% RSLogix 500 project T4150574.RSS, saved by version 8.10.00.18 %
PROJECT "T4150574"    % processor: SLC 500, 1747-L542 %

PROGRAM FILES
  LAD 2   89 rungs
  LAD 3   93 rungs
  LAD 4   69 rungs
  LAD 5   3 rungs
  LAD 6   136 rungs
  LAD 9   34 rungs
  LAD 10   90 rungs
  LAD 11   20 rungs
  LAD 12   13 rungs
  LAD 15   61 rungs
  LAD 16   27 rungs
  LAD 17   7 rungs
  LAD 18   55 rungs
  LAD 21   5 rungs
  LAD 22   82 rungs
  LAD 23   74 rungs
  LAD 24   136 rungs
  LAD 26   178 rungs
  LAD 27   27 rungs
  LAD 28   29 rungs
  LAD 31   238 rungs
  LAD 36   69 rungs
  LAD 41   9 rungs
  LAD 50   338 rungs
  LAD 51   183 rungs
  LAD 52   5 rungs
  LAD 53   6 rungs
  LAD 60   11 rungs
  LAD 71   9 rungs
  LAD 75   5 rungs
  LAD 76   5 rungs
  LAD 77   5 rungs
  LAD 78   6 rungs
  LAD 80   7 rungs
  LAD 120   43 rungs
  LAD 126   33 rungs
  LAD 127   30 rungs
  LAD 129   29 rungs
  LAD 131   44 rungs
  LAD 132   40 rungs
  LAD 133   25 rungs
  LAD 134   25 rungs

DATA FILES
  O0 OUTPUT  58 elements
  I1 INPUT  52 elements
  S2 STATUS  164 elements
  B3 BINARY  150 elements
  T4 TIMER  122 elements
  C5 COUNTER  6 elements
  R6 CONTROL  20 elements
  N7 INTEGER  53 elements
  F8 FLOAT  50 elements
  N9   14 elements
  B10   12 elements
  B11   33 elements
  B12   14 elements
  B15   1 elements
  B16   5 elements
  B17   5 elements
  B18   4 elements
  T21   85 elements
  B22   12 elements
  B23   8 elements
  B24   8 elements
  N25   195 elements
  B28   10 elements
  B29   15 elements
  B30   1 elements
  T31   50 elements
  N32   137 elements
  B35   9 elements
  B36   2 elements
  N40   240 elements
  N41   240 elements
  N42   240 elements
  N43   240 elements
  N44   240 elements
  N45   240 elements
  N46   240 elements
  N47   240 elements
  N48   120 elements
  B49   50 elements
  N50   60 elements
  N51   256 elements
  N52   100 elements
  B53   100 elements
  N54   100 elements
  N60   214 elements
  N61   250 elements
  N62   250 elements
  N63   250 elements
  N75   200 elements
  N76   50 elements
  N77   100 elements
  N78   50 elements
  N79   50 elements
  B84   4 elements
  N89   200 elements
  N90   20 elements
  N91   250 elements
  N92   250 elements
  N93   250 elements
  N94   250 elements
  N95   250 elements
  N100   50 elements
  N105   20 elements
  N110   80 elements

LADDER 2
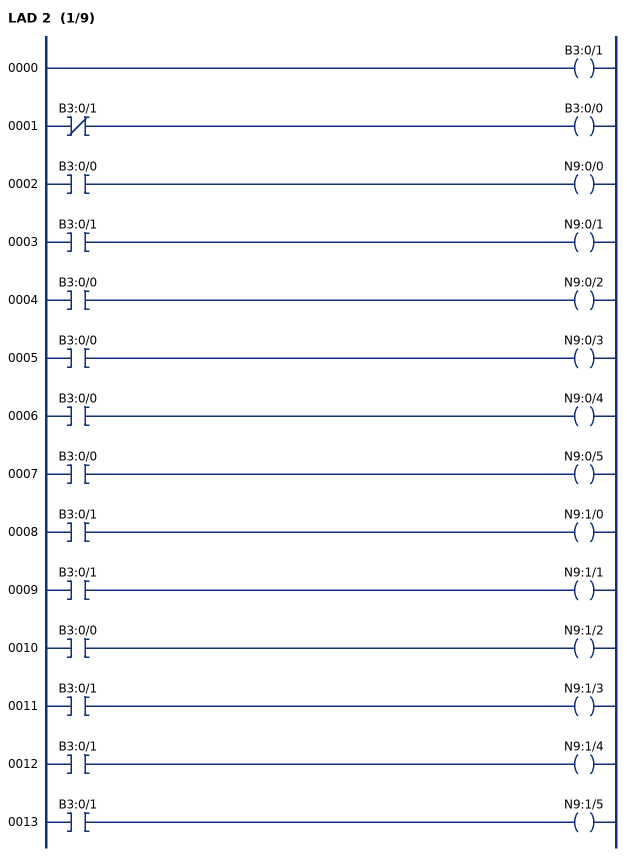
% Rung: 0 %
SOR OTE B3:0/1 EOR
% Rung: 1 %
SOR XIO B3:0/1 OTE B3:0/0 EOR
% Rung: 2 %
SOR XIC B3:0/0 OTE N9:0/0 EOR
% Rung: 3 %
SOR XIC B3:0/1 OTE N9:0/1 EOR
% Rung: 4 %
SOR XIC B3:0/0 OTE N9:0/2 EOR
% Rung: 5 %
SOR XIC B3:0/0 OTE N9:0/3 EOR
% Rung: 6 %
SOR XIC B3:0/0 OTE N9:0/4 EOR
% Rung: 7 %
SOR XIC B3:0/0 OTE N9:0/5 EOR
% Rung: 8 %
SOR XIC B3:0/1 OTE N9:1/0 EOR
% Rung: 9 %
SOR XIC B3:0/1 OTE N9:1/1 EOR
% Rung: 10 %
SOR XIC B3:0/0 OTE N9:1/2 EOR
% Rung: 11 %
SOR XIC B3:0/1 OTE N9:1/3 EOR
% Rung: 12 %
SOR XIC B3:0/1 OTE N9:1/4 EOR
% Rung: 13 %
SOR XIC B3:0/1 OTE N9:1/5 EOR

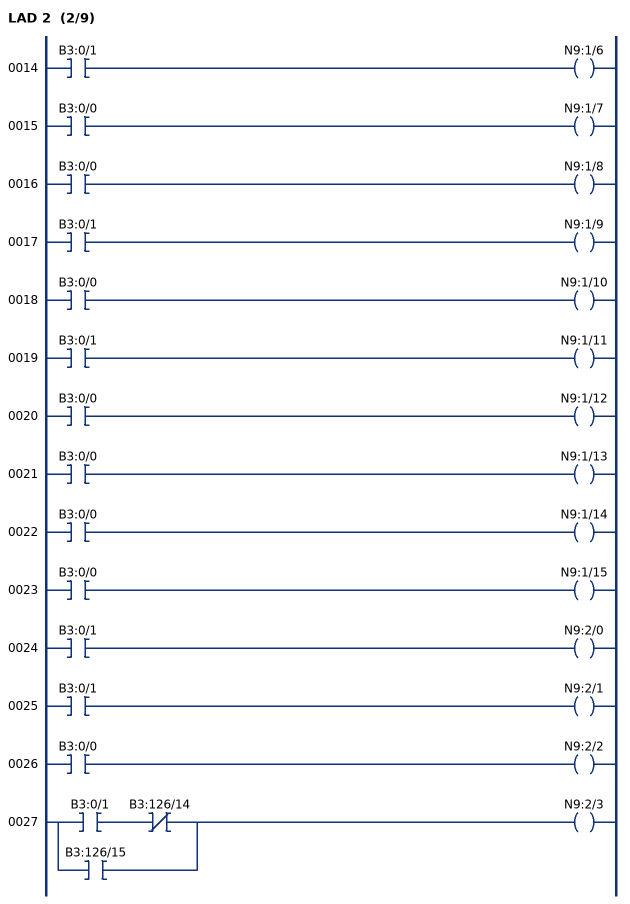
% Rung: 14 %
SOR XIC B3:0/1 OTE N9:1/6 EOR
% Rung: 15 %
SOR XIC B3:0/0 OTE N9:1/7 EOR
% Rung: 16 %
SOR XIC B3:0/0 OTE N9:1/8 EOR
% Rung: 17 %
SOR XIC B3:0/1 OTE N9:1/9 EOR
% Rung: 18 %
SOR XIC B3:0/0 OTE N9:1/10 EOR
% Rung: 19 %
SOR XIC B3:0/1 OTE N9:1/11 EOR
% Rung: 20 %
SOR XIC B3:0/0 OTE N9:1/12 EOR
% Rung: 21 %
SOR XIC B3:0/0 OTE N9:1/13 EOR
% Rung: 22 %
SOR XIC B3:0/0 OTE N9:1/14 EOR
% Rung: 23 %
SOR XIC B3:0/0 OTE N9:1/15 EOR
% Rung: 24 %
SOR XIC B3:0/1 OTE N9:2/0 EOR
% Rung: 25 %
SOR XIC B3:0/1 OTE N9:2/1 EOR
% Rung: 26 %
SOR XIC B3:0/0 OTE N9:2/2 EOR
% Rung: 27 %
SOR BST XIC B3:0/1 XIO B3:126/14 NXB XIC B3:126/15 BND OTE N9:2/3 EOR

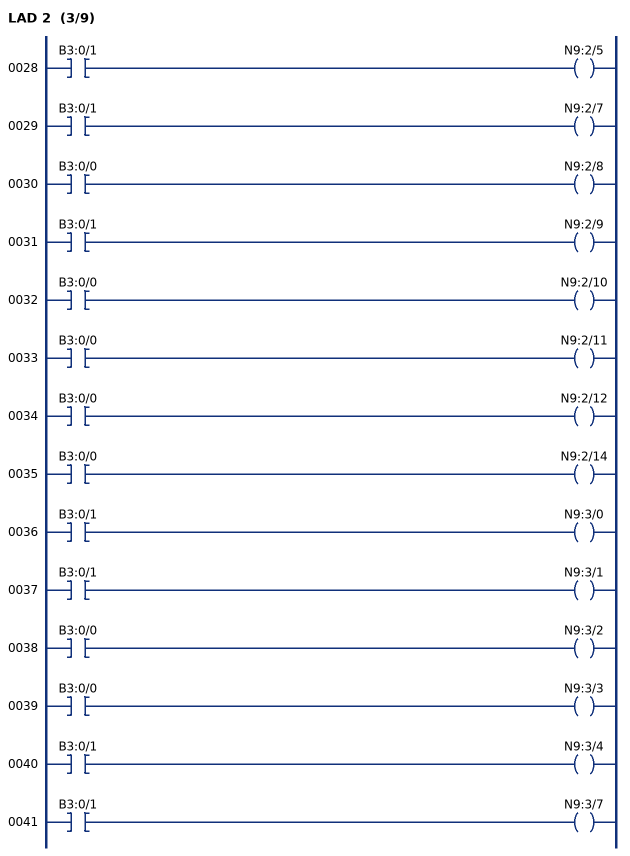
% Rung: 28 %
SOR XIC B3:0/1 OTE N9:2/5 EOR
% Rung: 29 %
SOR XIC B3:0/1 OTE N9:2/7 EOR
% Rung: 30 %
SOR XIC B3:0/0 OTE N9:2/8 EOR
% Rung: 31 %
SOR XIC B3:0/1 OTE N9:2/9 EOR
% Rung: 32 %
SOR XIC B3:0/0 OTE N9:2/10 EOR
% Rung: 33 %
SOR XIC B3:0/0 OTE N9:2/11 EOR
% Rung: 34 %
SOR XIC B3:0/0 OTE N9:2/12 EOR
% Rung: 35 %
SOR XIC B3:0/0 OTE N9:2/14 EOR
% Rung: 36 %
SOR XIC B3:0/1 OTE N9:3/0 EOR
% Rung: 37 %
SOR XIC B3:0/1 OTE N9:3/1 EOR
% Rung: 38 %
SOR XIC B3:0/0 OTE N9:3/2 EOR
% Rung: 39 %
SOR XIC B3:0/0 OTE N9:3/3 EOR
% Rung: 40 %
SOR XIC B3:0/1 OTE N9:3/4 EOR
% Rung: 41 %
SOR XIC B3:0/1 OTE N9:3/7 EOR

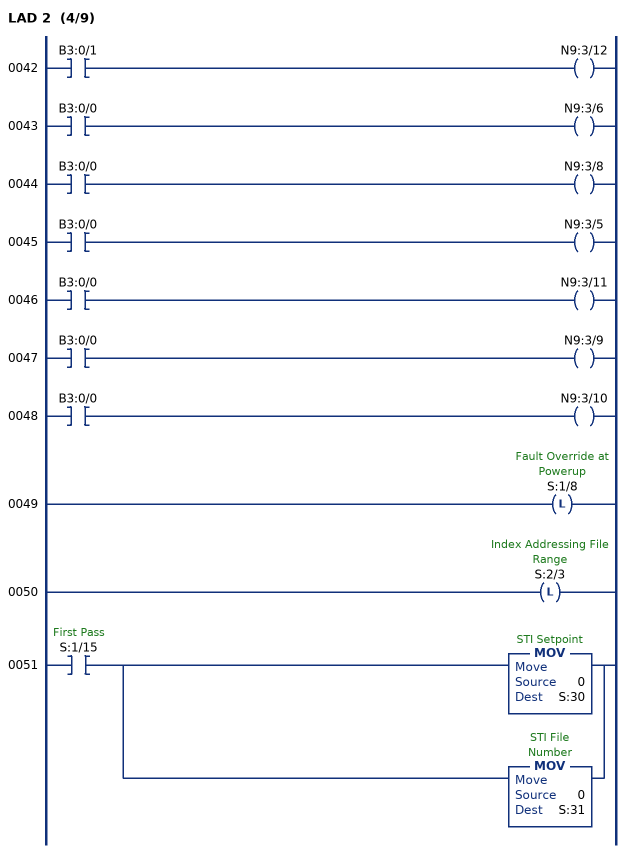
% Rung: 42 %
SOR XIC B3:0/1 OTE N9:3/12 EOR
% Rung: 43 %
SOR XIC B3:0/0 OTE N9:3/6 EOR
% Rung: 44 %
SOR XIC B3:0/0 OTE N9:3/8 EOR
% Rung: 45 %
SOR XIC B3:0/0 OTE N9:3/5 EOR
% Rung: 46 %
SOR XIC B3:0/0 OTE N9:3/11 EOR
% Rung: 47 %
SOR XIC B3:0/0 OTE N9:3/9 EOR
% Rung: 48 %
SOR XIC B3:0/0 OTE N9:3/10 EOR
% Rung: 49 %
SOR OTL S:1/8 EOR
%   S:1/8  "Fault Override at Powerup" %
% Rung: 50 %
SOR OTL S:2/3 EOR
%   S:2/3  "Index Addressing File Range" %
% Rung: 51 %
SOR XIC S:1/15 BST MOV 0 S:30 NXB MOV 0 S:31 BND EOR
%   S:1/15  "First Pass" %
%   S:30  "STI Setpoint" %
%   S:31  "STI File Number" %

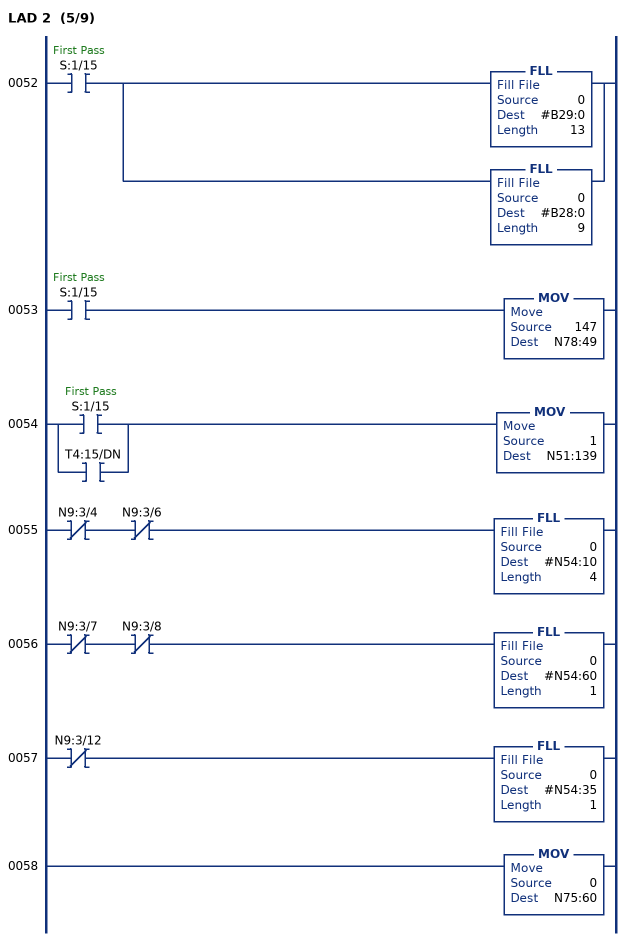
% Rung: 52 %
SOR XIC S:1/15 BST FLL 0 #B29:0 13 NXB FLL 0 #B28:0 9 BND EOR
%   S:1/15  "First Pass" %
% Rung: 53 %
SOR XIC S:1/15 MOV 147 N78:49 EOR
%   S:1/15  "First Pass" %
% Rung: 54 %
SOR BST XIC S:1/15 NXB XIC T4:15/DN BND MOV 1 N51:139 EOR
%   S:1/15  "First Pass" %
% Rung: 55 %
SOR XIO N9:3/4 XIO N9:3/6 FLL 0 #N54:10 4 EOR
% Rung: 56 %
SOR XIO N9:3/7 XIO N9:3/8 FLL 0 #N54:60 1 EOR
% Rung: 57 %
SOR XIO N9:3/12 FLL 0 #N54:35 1 EOR
% Rung: 58 %
SOR MOV 0 N75:60 EOR

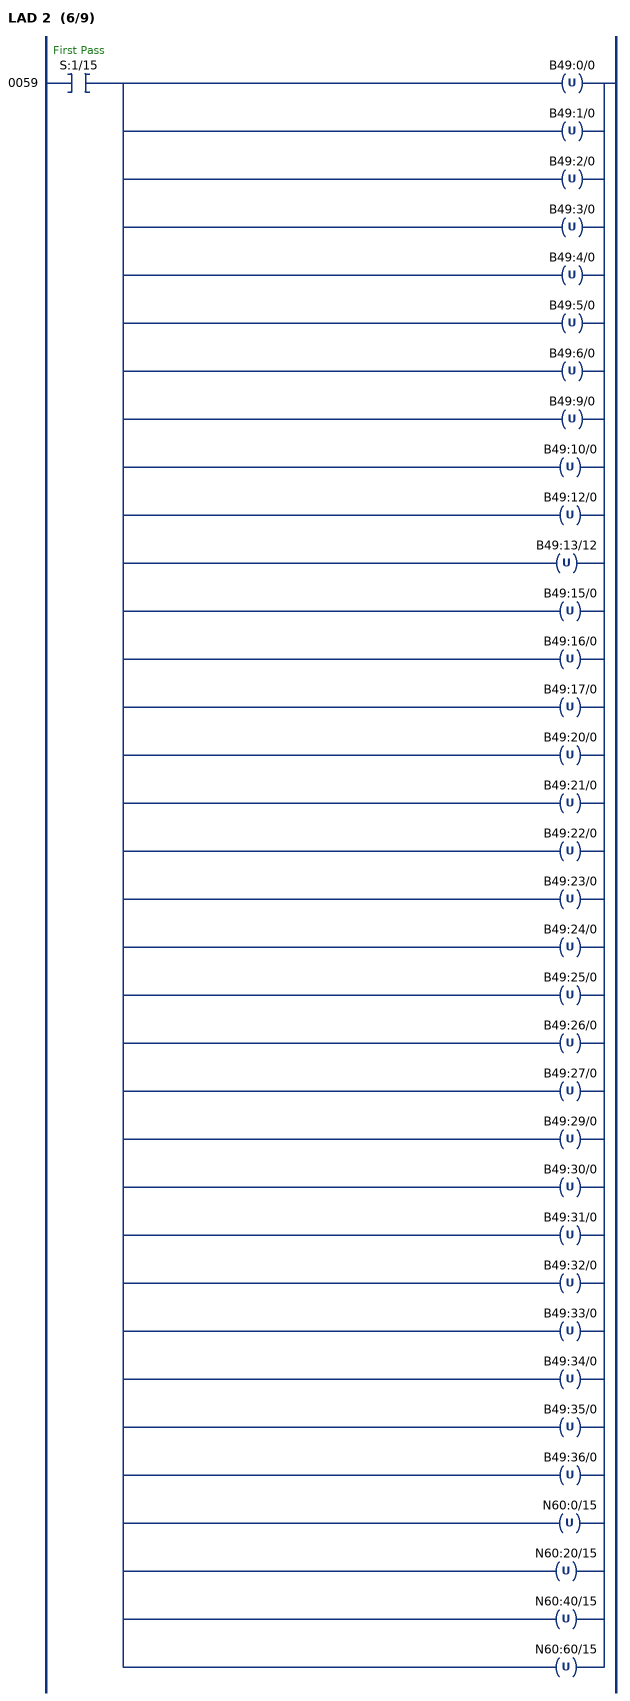
% Rung: 59 %
SOR XIC S:1/15 BST OTU B49:0/0 NXB OTU B49:1/0 NXB OTU B49:2/0 NXB OTU B49:3/0 NXB OTU B49:4/0 NXB OTU B49:5/0 NXB OTU B49:6/0 NXB OTU B49:9/0 NXB OTU B49:10/0 NXB OTU B49:12/0 NXB OTU B49:13/12 NXB OTU B49:15/0 NXB OTU B49:16/0 NXB OTU B49:17/0 NXB OTU B49:20/0 NXB OTU B49:21/0 NXB OTU B49:22/0 NXB OTU B49:23/0 NXB OTU B49:24/0 NXB OTU B49:25/0 NXB OTU B49:26/0 NXB OTU B49:27/0 NXB OTU B49:29/0 NXB OTU B49:30/0 NXB OTU B49:31/0 NXB OTU B49:32/0 NXB OTU B49:33/0 NXB OTU B49:34/0 NXB OTU B49:35/0 NXB OTU B49:36/0 NXB OTU N60:0/15 NXB OTU N60:20/15 NXB OTU N60:40/15 NXB OTU N60:60/15 BND EOR
%   S:1/15  "First Pass" %

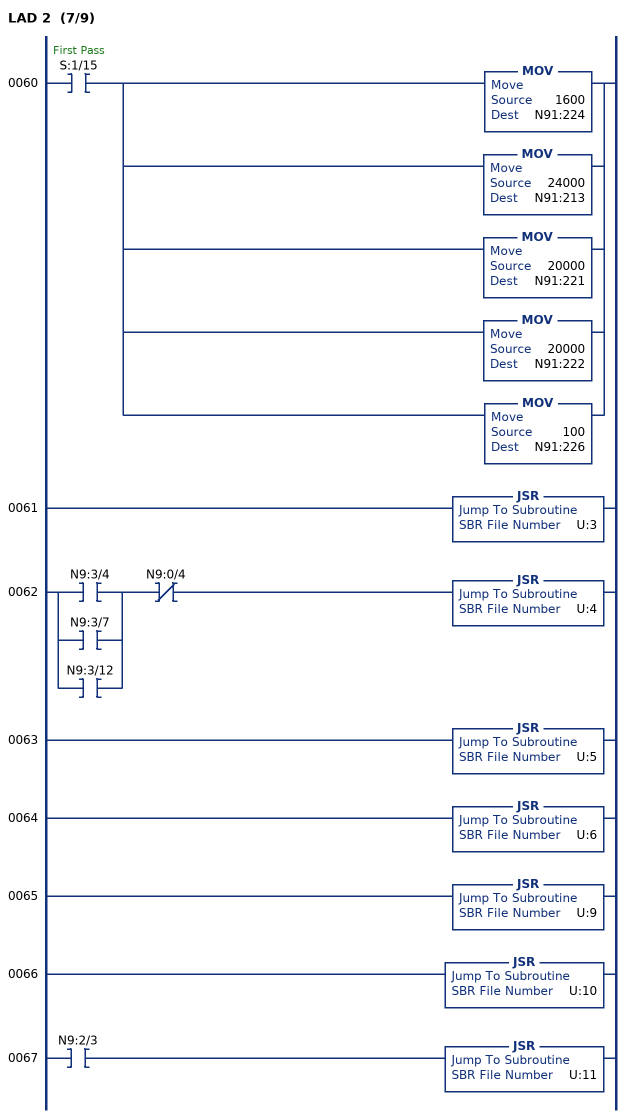
% Rung: 60 %
SOR XIC S:1/15 BST MOV 1600 N91:224 NXB MOV 24000 N91:213 NXB MOV 20000 N91:221 NXB MOV 20000 N91:222 NXB MOV 100 N91:226 BND EOR
%   S:1/15  "First Pass" %
% Rung: 61 %
SOR JSR U:3 EOR
% Rung: 62 %
SOR BST XIC N9:3/4 NXB XIC N9:3/7 NXB XIC N9:3/12 BND XIO N9:0/4 JSR U:4 EOR
% Rung: 63 %
SOR JSR U:5 EOR
% Rung: 64 %
SOR JSR U:6 EOR
% Rung: 65 %
SOR JSR U:9 EOR
% Rung: 66 %
SOR JSR U:10 EOR
% Rung: 67 %
SOR XIC N9:2/3 JSR U:11 EOR

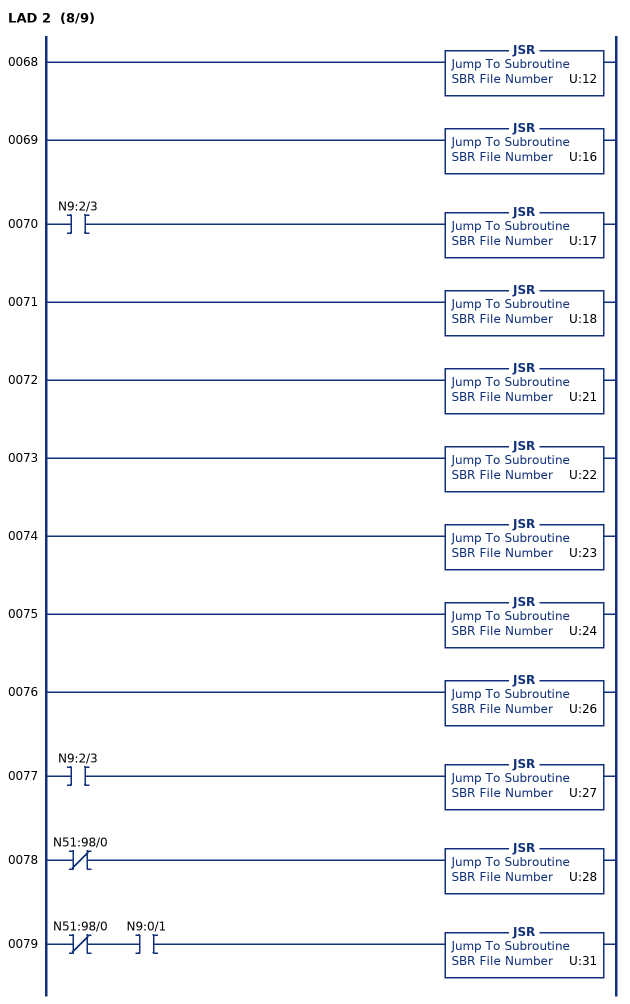
% Rung: 68 %
SOR JSR U:12 EOR
% Rung: 69 %
SOR JSR U:16 EOR
% Rung: 70 %
SOR XIC N9:2/3 JSR U:17 EOR
% Rung: 71 %
SOR JSR U:18 EOR
% Rung: 72 %
SOR JSR U:21 EOR
% Rung: 73 %
SOR JSR U:22 EOR
% Rung: 74 %
SOR JSR U:23 EOR
% Rung: 75 %
SOR JSR U:24 EOR
% Rung: 76 %
SOR JSR U:26 EOR
% Rung: 77 %
SOR XIC N9:2/3 JSR U:27 EOR
% Rung: 78 %
SOR XIO N51:98/0 JSR U:28 EOR
% Rung: 79 %
SOR XIO N51:98/0 XIC N9:0/1 JSR U:31 EOR

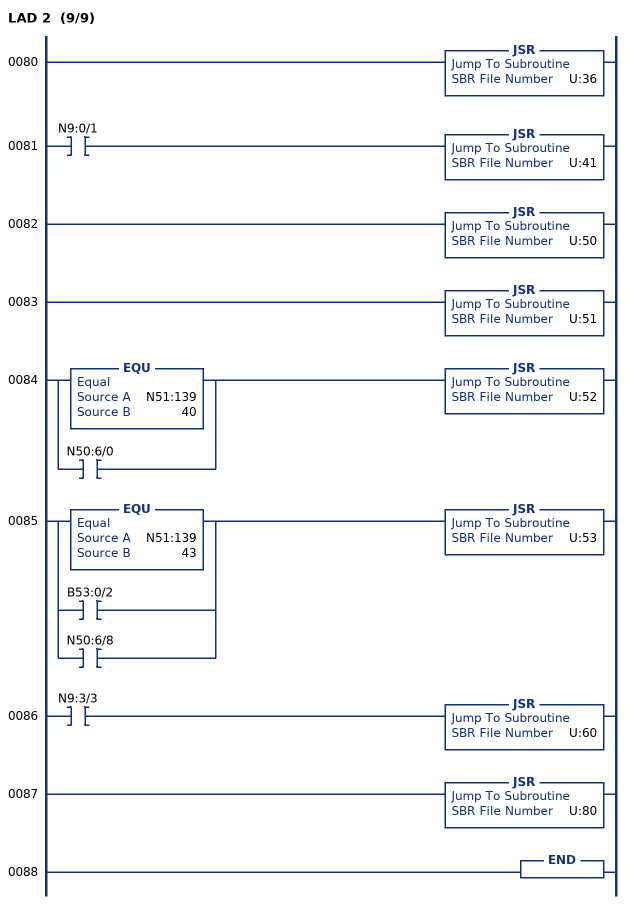
% Rung: 80 %
SOR JSR U:36 EOR
% Rung: 81 %
SOR XIC N9:0/1 JSR U:41 EOR
% Rung: 82 %
SOR JSR U:50 EOR
% Rung: 83 %
SOR JSR U:51 EOR
% Rung: 84 %
SOR BST EQU N51:139 40 NXB XIC N50:6/0 BND JSR U:52 EOR
% Rung: 85 %
SOR BST EQU N51:139 43 NXB XIC B53:0/2 NXB XIC N50:6/8 BND JSR U:53 EOR
% Rung: 86 %
SOR XIC N9:3/3 JSR U:60 EOR
% Rung: 87 %
SOR JSR U:80 EOR
% Rung: 88 %
SOR END EOR

LADDER 3
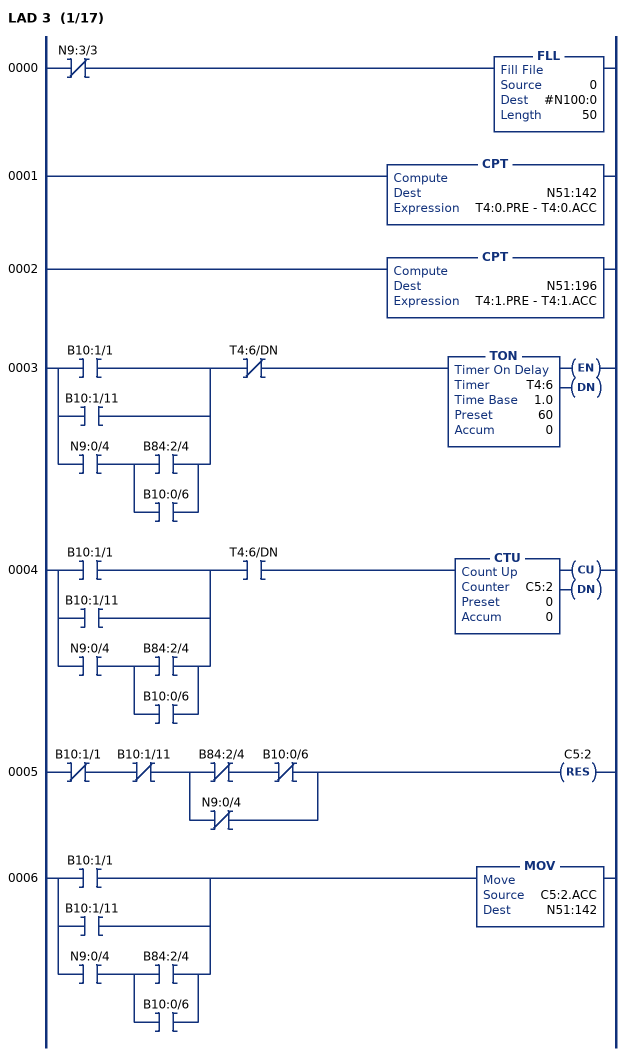
% Rung: 0 %
SOR XIO N9:3/3 FLL 0 #N100:0 50 EOR
% Rung: 1 %
SOR CPT N51:142 " T4:0.PRE - T4:0.ACC " EOR
% Rung: 2 %
SOR CPT N51:196 " T4:1.PRE - T4:1.ACC " EOR
% Rung: 3 %
SOR BST XIC B10:1/1 NXB XIC B10:1/11 NXB XIC N9:0/4 BST XIC B84:2/4 NXB XIC B10:0/6 BND BND XIO T4:6/DN TON T4:6 1.0 60 0 EOR
% Rung: 4 %
SOR BST XIC B10:1/1 NXB XIC B10:1/11 NXB XIC N9:0/4 BST XIC B84:2/4 NXB XIC B10:0/6 BND BND XIC T4:6/DN CTU C5:2 0 0 EOR
% Rung: 5 %
SOR XIO B10:1/1 XIO B10:1/11 BST XIO B84:2/4 XIO B10:0/6 NXB XIO N9:0/4 BND RES C5:2 EOR
% Rung: 6 %
SOR BST XIC B10:1/1 NXB XIC B10:1/11 NXB XIC N9:0/4 BST XIC B84:2/4 NXB XIC B10:0/6 BND BND MOV C5:2.ACC N51:142 EOR

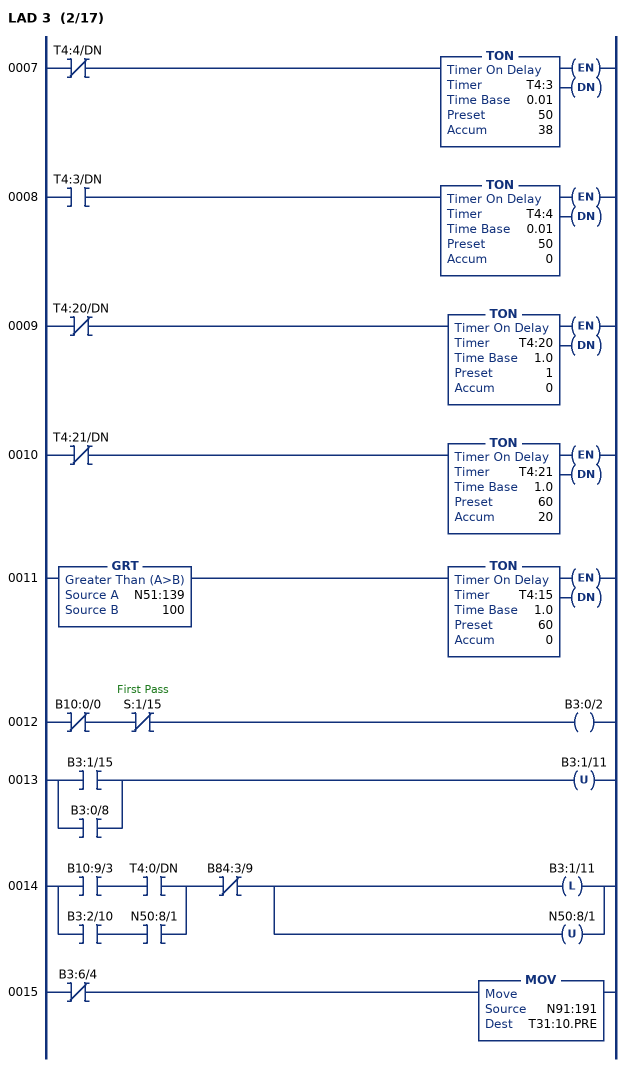
% Rung: 7 %
SOR XIO T4:4/DN TON T4:3 0.01 50 38 EOR
% Rung: 8 %
SOR XIC T4:3/DN TON T4:4 0.01 50 0 EOR
% Rung: 9 %
SOR XIO T4:20/DN TON T4:20 1.0 1 0 EOR
% Rung: 10 %
SOR XIO T4:21/DN TON T4:21 1.0 60 20 EOR
% Rung: 11 %
SOR GRT N51:139 100 TON T4:15 1.0 60 0 EOR
% Rung: 12 %
SOR XIO B10:0/0 XIO S:1/15 OTE B3:0/2 EOR
%   S:1/15  "First Pass" %
% Rung: 13 %
SOR BST XIC B3:1/15 NXB XIC B3:0/8 BND OTU B3:1/11 EOR
% Rung: 14 %
SOR BST XIC B10:9/3 XIC T4:0/DN NXB XIC B3:2/10 XIC N50:8/1 BND XIO B84:3/9 BST OTL B3:1/11 NXB OTU N50:8/1 BND EOR
% Rung: 15 %
SOR XIO B3:6/4 MOV N91:191 T31:10.PRE EOR

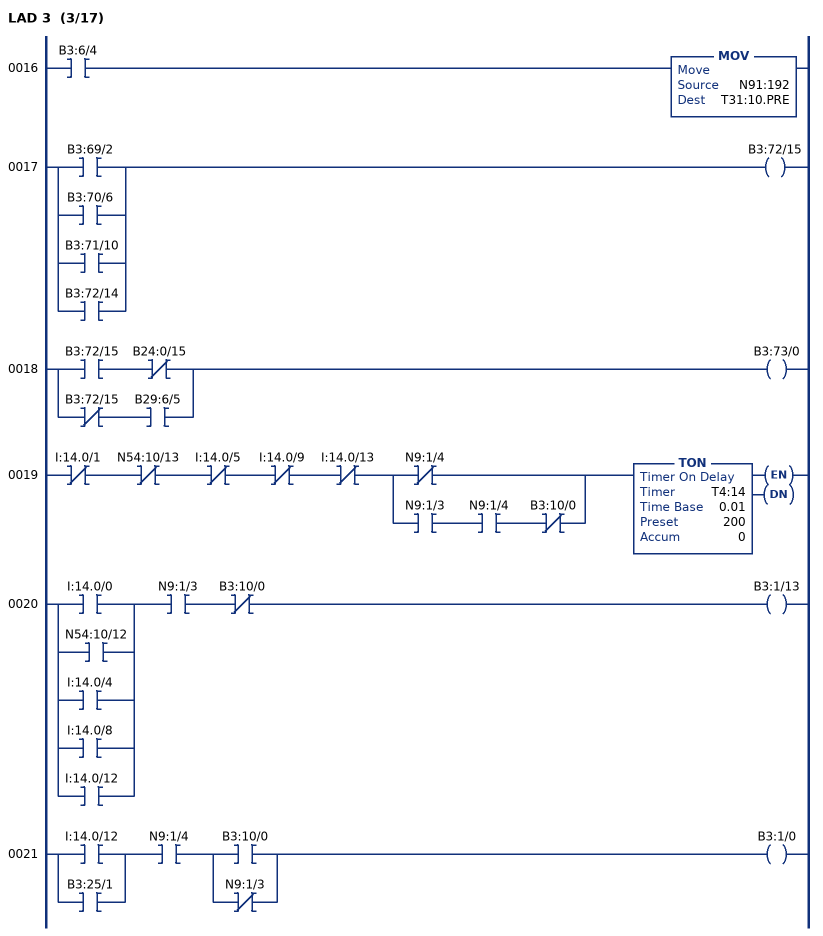
% Rung: 16 %
SOR XIC B3:6/4 MOV N91:192 T31:10.PRE EOR
% Rung: 17 %
SOR BST XIC B3:69/2 NXB XIC B3:70/6 NXB XIC B3:71/10 NXB XIC B3:72/14 BND OTE B3:72/15 EOR
% Rung: 18 %
SOR BST XIC B3:72/15 XIO B24:0/15 NXB XIO B3:72/15 XIC B29:6/5 BND OTE B3:73/0 EOR
% Rung: 19 %
SOR XIO I:14.0/1 XIO N54:10/13 XIO I:14.0/5 XIO I:14.0/9 XIO I:14.0/13 BST XIO N9:1/4 NXB XIC N9:1/3 XIC N9:1/4 XIO B3:10/0 BND TON T4:14 0.01 200 0 EOR
% Rung: 20 %
SOR BST BST XIC I:14.0/0 NXB XIC N54:10/12 BND NXB XIC I:14.0/4 NXB XIC I:14.0/8 NXB XIC I:14.0/12 BND XIC N9:1/3 XIO B3:10/0 OTE B3:1/13 EOR
% Rung: 21 %
SOR BST XIC I:14.0/12 NXB XIC B3:25/1 BND XIC N9:1/4 BST XIC B3:10/0 NXB XIO N9:1/3 BND OTE B3:1/0 EOR

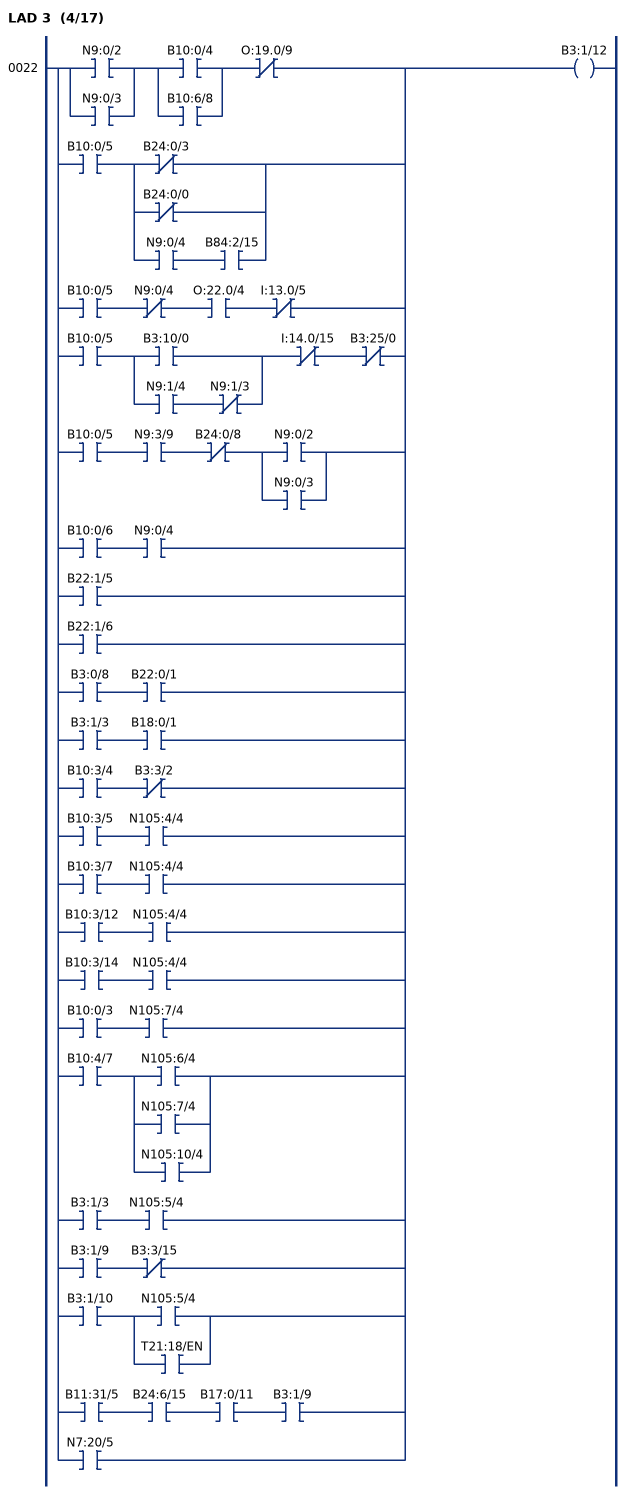
% Rung: 22 %
SOR BST BST XIC N9:0/2 NXB XIC N9:0/3 BND BST XIC B10:0/4 NXB XIC B10:6/8 BND XIO O:19.0/9 NXB XIC B10:0/5 BST XIO B24:0/3 NXB XIO B24:0/0 NXB XIC N9:0/4 XIC B84:2/15 BND NXB XIC B10:0/5 XIO N9:0/4 XIC O:22.0/4 XIO I:13.0/5 NXB XIC B10:0/5 BST XIC B3:10/0 NXB XIC N9:1/4 XIO N9:1/3 BND XIO I:14.0/15 XIO B3:25/0 NXB XIC B10:0/5 XIC N9:3/9 XIO B24:0/8 BST XIC N9:0/2 NXB XIC N9:0/3 BND NXB XIC B10:0/6 XIC N9:0/4 NXB XIC B22:1/5 NXB XIC B22:1/6 NXB XIC B3:0/8 XIC B22:0/1 NXB XIC B3:1/3 XIC B18:0/1 NXB XIC B10:3/4 XIO B3:3/2 NXB XIC B10:3/5 XIC N105:4/4 NXB XIC B10:3/7 XIC N105:4/4 NXB XIC B10:3/12 XIC N105:4/4 NXB XIC B10:3/14 XIC N105:4/4 NXB XIC B10:0/3 XIC N105:7/4 NXB XIC B10:4/7 BST XIC N105:6/4 NXB XIC N105:7/4 NXB XIC N105:10/4 BND NXB XIC B3:1/3 XIC N105:5/4 NXB XIC B3:1/9 XIO B3:3/15 NXB XIC B3:1/10 BST XIC N105:5/4 NXB XIC T21:18/EN BND NXB XIC B11:31/5 XIC B24:6/15 XIC B17:0/11 XIC B3:1/9 NXB XIC N7:20/5 BND OTE B3:1/12 EOR

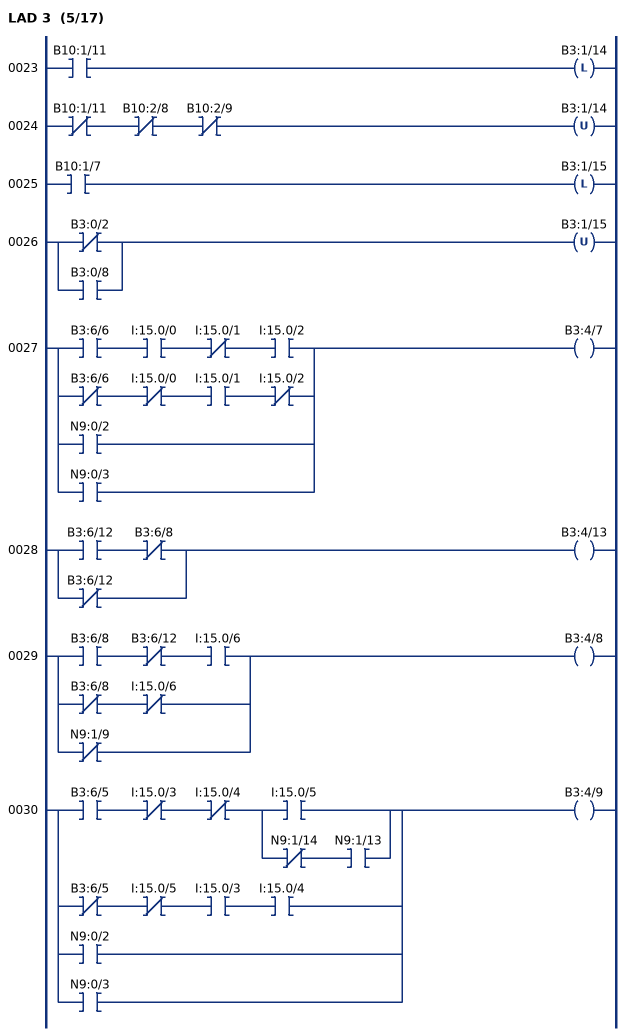
% Rung: 23 %
SOR XIC B10:1/11 OTL B3:1/14 EOR
% Rung: 24 %
SOR XIO B10:1/11 XIO B10:2/8 XIO B10:2/9 OTU B3:1/14 EOR
% Rung: 25 %
SOR XIC B10:1/7 OTL B3:1/15 EOR
% Rung: 26 %
SOR BST XIO B3:0/2 NXB XIC B3:0/8 BND OTU B3:1/15 EOR
% Rung: 27 %
SOR BST XIC B3:6/6 XIC I:15.0/0 XIO I:15.0/1 XIC I:15.0/2 NXB XIO B3:6/6 XIO I:15.0/0 XIC I:15.0/1 XIO I:15.0/2 NXB XIC N9:0/2 NXB XIC N9:0/3 BND OTE B3:4/7 EOR
% Rung: 28 %
SOR BST XIC B3:6/12 XIO B3:6/8 NXB XIO B3:6/12 BND OTE B3:4/13 EOR
% Rung: 29 %
SOR BST XIC B3:6/8 XIO B3:6/12 XIC I:15.0/6 NXB XIO B3:6/8 XIO I:15.0/6 NXB XIO N9:1/9 BND OTE B3:4/8 EOR
% Rung: 30 %
SOR BST XIC B3:6/5 XIO I:15.0/3 XIO I:15.0/4 BST XIC I:15.0/5 NXB XIO N9:1/14 XIC N9:1/13 BND NXB XIO B3:6/5 XIO I:15.0/5 XIC I:15.0/3 XIC I:15.0/4 NXB XIC N9:0/2 NXB XIC N9:0/3 BND OTE B3:4/9 EOR

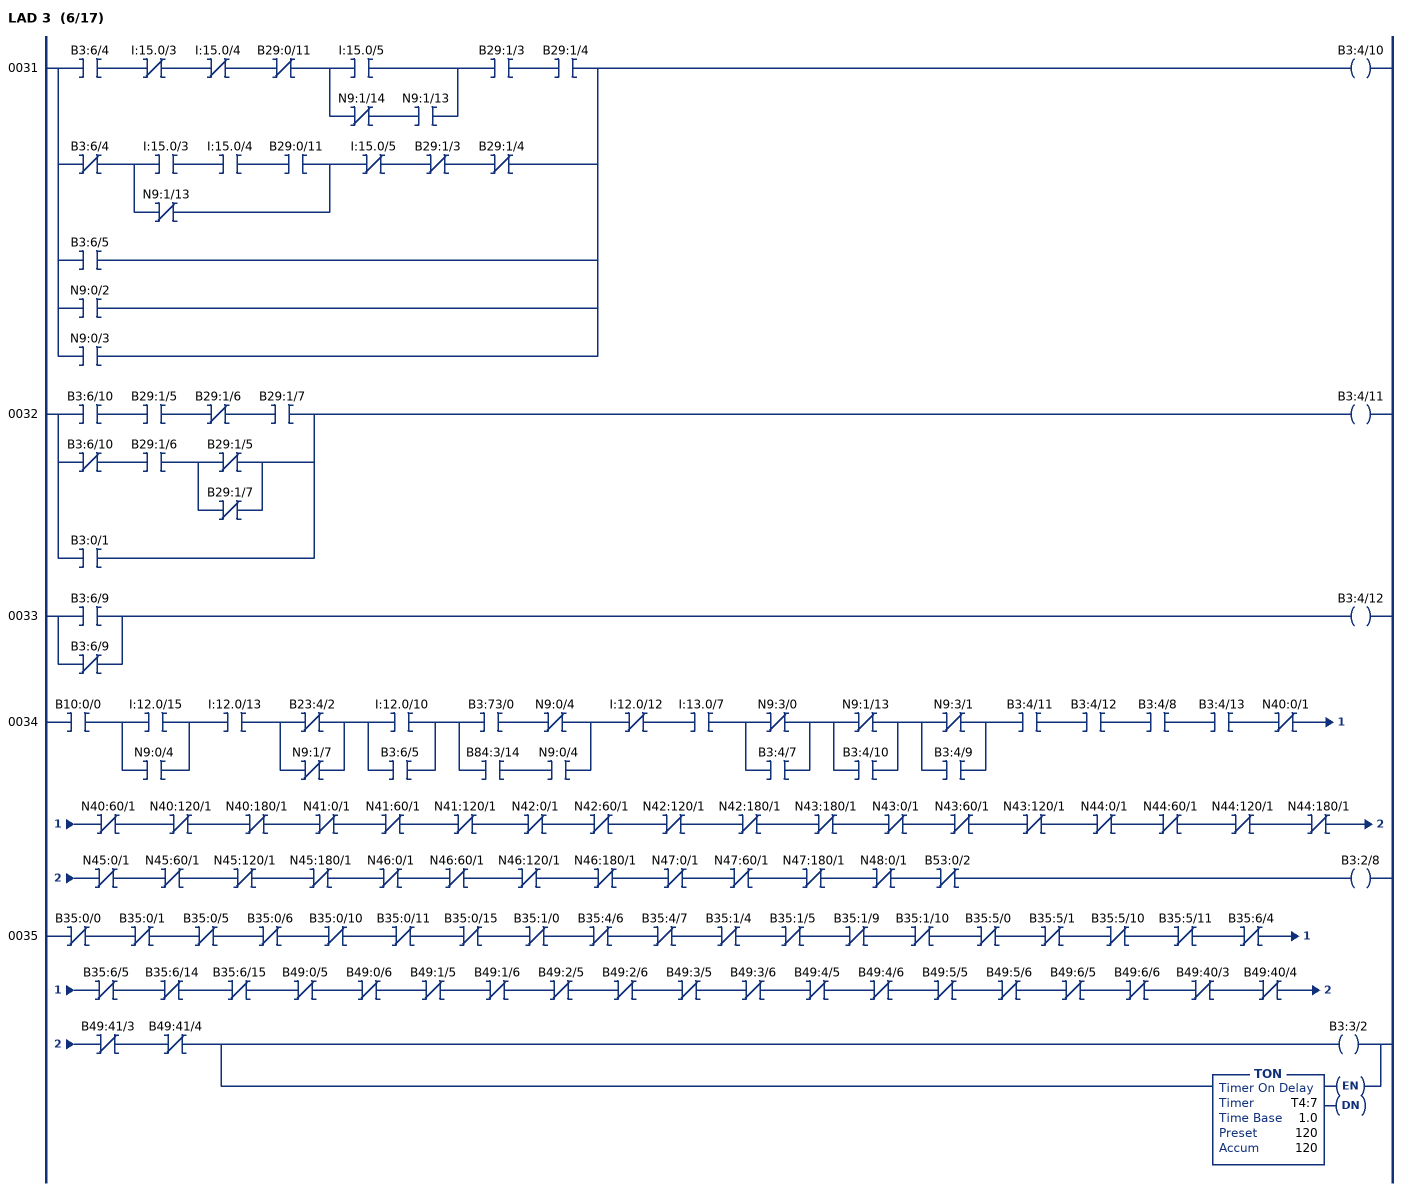
% Rung: 31 %
SOR BST XIC B3:6/4 XIO I:15.0/3 XIO I:15.0/4 XIO B29:0/11 BST XIC I:15.0/5 NXB XIO N9:1/14 XIC N9:1/13 BND XIC B29:1/3 XIC B29:1/4 NXB XIO B3:6/4 BST XIC I:15.0/3 XIC I:15.0/4 XIC B29:0/11 NXB XIO N9:1/13 BND XIO I:15.0/5 XIO B29:1/3 XIO B29:1/4 NXB XIC B3:6/5 NXB XIC N9:0/2 NXB XIC N9:0/3 BND OTE B3:4/10 EOR
% Rung: 32 %
SOR BST XIC B3:6/10 XIC B29:1/5 XIO B29:1/6 XIC B29:1/7 NXB XIO B3:6/10 XIC B29:1/6 BST XIO B29:1/5 NXB XIO B29:1/7 BND NXB XIC B3:0/1 BND OTE B3:4/11 EOR
% Rung: 33 %
SOR BST XIC B3:6/9 NXB XIO B3:6/9 BND OTE B3:4/12 EOR
% Rung: 34 %
SOR XIC B10:0/0 BST XIC I:12.0/15 NXB XIC N9:0/4 BND XIC I:12.0/13 BST XIO B23:4/2 NXB XIO N9:1/7 BND BST XIC I:12.0/10 NXB XIC B3:6/5 BND BST XIC B3:73/0 XIO N9:0/4 NXB XIC B84:3/14 XIC N9:0/4 BND XIO I:12.0/12 XIC I:13.0/7 BST XIO N9:3/0 NXB XIC B3:4/7 BND BST XIO N9:1/13 NXB XIC B3:4/10 BND BST XIO N9:3/1 NXB XIC B3:4/9 BND XIC B3:4/11 XIC B3:4/12 XIC B3:4/8 XIC B3:4/13 XIO N40:0/1 XIO N40:60/1 XIO N40:120/1 XIO N40:180/1 XIO N41:0/1 XIO N41:60/1 XIO N41:120/1 XIO N42:0/1 XIO N42:60/1 XIO N42:120/1 XIO N42:180/1 XIO N43:180/1 XIO N43:0/1 XIO N43:60/1 XIO N43:120/1 XIO N44:0/1 XIO N44:60/1 XIO N44:120/1 XIO N44:180/1 XIO N45:0/1 XIO N45:60/1 XIO N45:120/1 XIO N45:180/1 XIO N46:0/1 XIO N46:60/1 XIO N46:120/1 XIO N46:180/1 XIO N47:0/1 XIO N47:60/1 XIO N47:180/1 XIO N48:0/1 XIO B53:0/2 OTE B3:2/8 EOR
% Rung: 35 %
SOR XIO B35:0/0 XIO B35:0/1 XIO B35:0/5 XIO B35:0/6 XIO B35:0/10 XIO B35:0/11 XIO B35:0/15 XIO B35:1/0 XIO B35:4/6 XIO B35:4/7 XIO B35:1/4 XIO B35:1/5 XIO B35:1/9 XIO B35:1/10 XIO B35:5/0 XIO B35:5/1 XIO B35:5/10 XIO B35:5/11 XIO B35:6/4 XIO B35:6/5 XIO B35:6/14 XIO B35:6/15 XIO B49:0/5 XIO B49:0/6 XIO B49:1/5 XIO B49:1/6 XIO B49:2/5 XIO B49:2/6 XIO B49:3/5 XIO B49:3/6 XIO B49:4/5 XIO B49:4/6 XIO B49:5/5 XIO B49:5/6 XIO B49:6/5 XIO B49:6/6 XIO B49:40/3 XIO B49:40/4 XIO B49:41/3 XIO B49:41/4 BST OTE B3:3/2 NXB TON T4:7 1.0 120 120 BND EOR

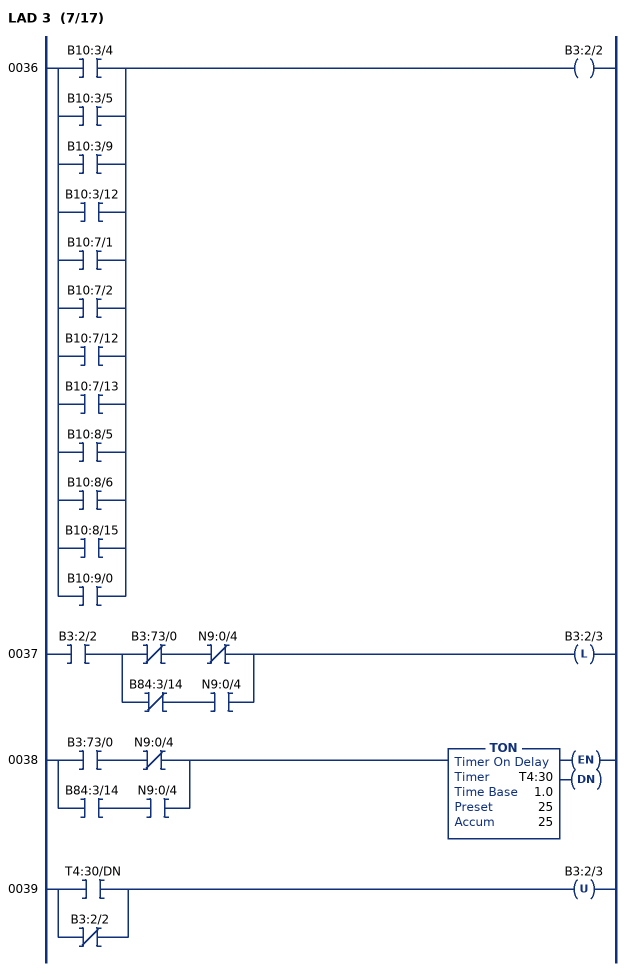
% Rung: 36 %
SOR BST XIC B10:3/4 NXB XIC B10:3/5 NXB XIC B10:3/9 NXB XIC B10:3/12 NXB XIC B10:7/1 NXB XIC B10:7/2 NXB XIC B10:7/12 NXB XIC B10:7/13 NXB XIC B10:8/5 NXB XIC B10:8/6 NXB XIC B10:8/15 NXB XIC B10:9/0 BND OTE B3:2/2 EOR
% Rung: 37 %
SOR XIC B3:2/2 BST XIO B3:73/0 XIO N9:0/4 NXB XIO B84:3/14 XIC N9:0/4 BND OTL B3:2/3 EOR
% Rung: 38 %
SOR BST XIC B3:73/0 XIO N9:0/4 NXB XIC B84:3/14 XIC N9:0/4 BND TON T4:30 1.0 25 25 EOR
% Rung: 39 %
SOR BST XIC T4:30/DN NXB XIO B3:2/2 BND OTU B3:2/3 EOR

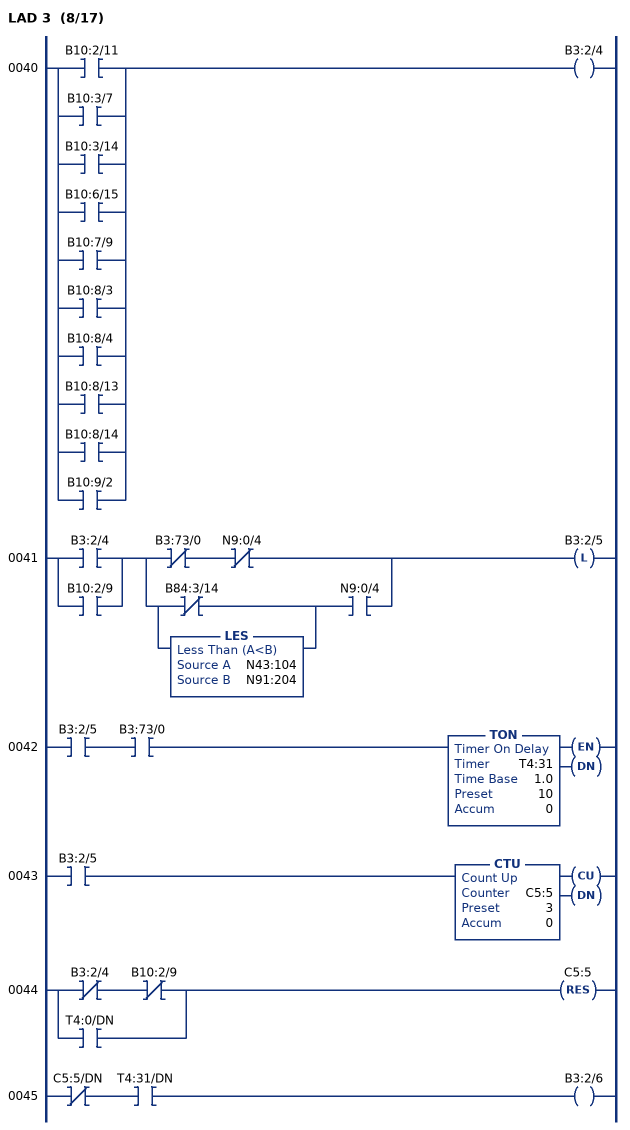
% Rung: 40 %
SOR BST XIC B10:2/11 NXB XIC B10:3/7 NXB XIC B10:3/14 NXB XIC B10:6/15 NXB XIC B10:7/9 NXB XIC B10:8/3 NXB XIC B10:8/4 NXB XIC B10:8/13 NXB XIC B10:8/14 NXB XIC B10:9/2 BND OTE B3:2/4 EOR
% Rung: 41 %
SOR BST XIC B3:2/4 NXB XIC B10:2/9 BND BST XIO B3:73/0 XIO N9:0/4 NXB BST XIO B84:3/14 NXB LES N43:104 N91:204 BND XIC N9:0/4 BND OTL B3:2/5 EOR
% Rung: 42 %
SOR XIC B3:2/5 XIC B3:73/0 TON T4:31 1.0 10 0 EOR
% Rung: 43 %
SOR XIC B3:2/5 CTU C5:5 3 0 EOR
% Rung: 44 %
SOR BST XIO B3:2/4 XIO B10:2/9 NXB XIC T4:0/DN BND RES C5:5 EOR
% Rung: 45 %
SOR XIO C5:5/DN XIC T4:31/DN OTE B3:2/6 EOR

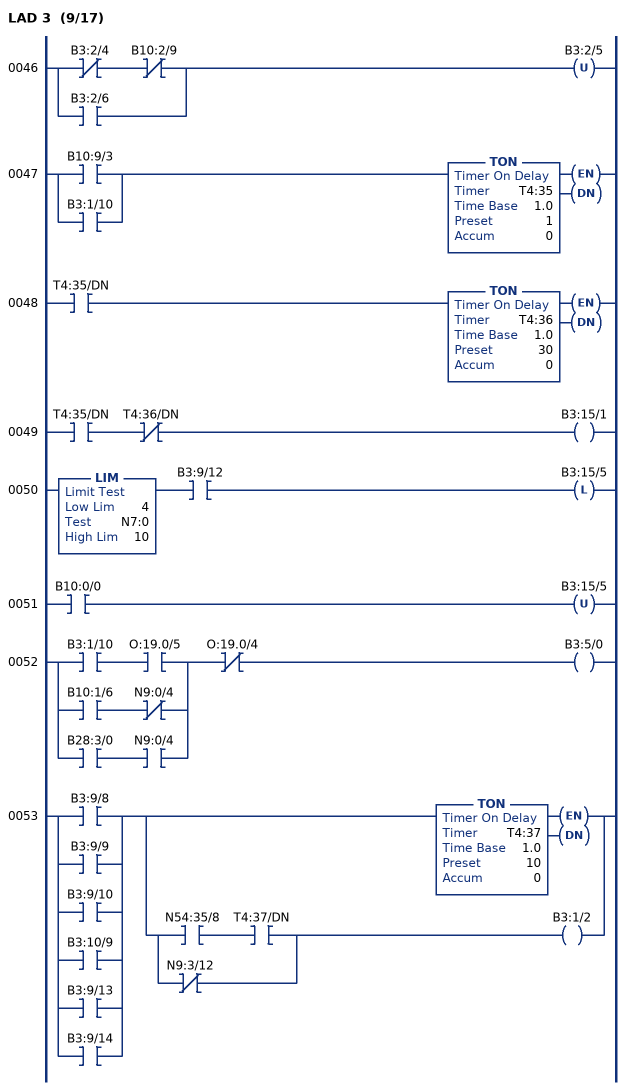
% Rung: 46 %
SOR BST XIO B3:2/4 XIO B10:2/9 NXB XIC B3:2/6 BND OTU B3:2/5 EOR
% Rung: 47 %
SOR BST XIC B10:9/3 NXB XIC B3:1/10 BND TON T4:35 1.0 1 0 EOR
% Rung: 48 %
SOR XIC T4:35/DN TON T4:36 1.0 30 0 EOR
% Rung: 49 %
SOR XIC T4:35/DN XIO T4:36/DN OTE B3:15/1 EOR
% Rung: 50 %
SOR LIM 4 N7:0 10 XIC B3:9/12 OTL B3:15/5 EOR
% Rung: 51 %
SOR XIC B10:0/0 OTU B3:15/5 EOR
% Rung: 52 %
SOR BST XIC B3:1/10 XIC O:19.0/5 NXB XIC B10:1/6 XIO N9:0/4 NXB XIC B28:3/0 XIC N9:0/4 BND XIO O:19.0/4 OTE B3:5/0 EOR
% Rung: 53 %
SOR BST BST XIC B3:9/8 NXB XIC B3:9/9 NXB XIC B3:9/10 NXB XIC B3:10/9 BND NXB XIC B3:9/13 NXB XIC B3:9/14 BND BST TON T4:37 1.0 10 0 NXB BST XIC N54:35/8 XIC T4:37/DN NXB XIO N9:3/12 BND OTE B3:1/2 BND EOR

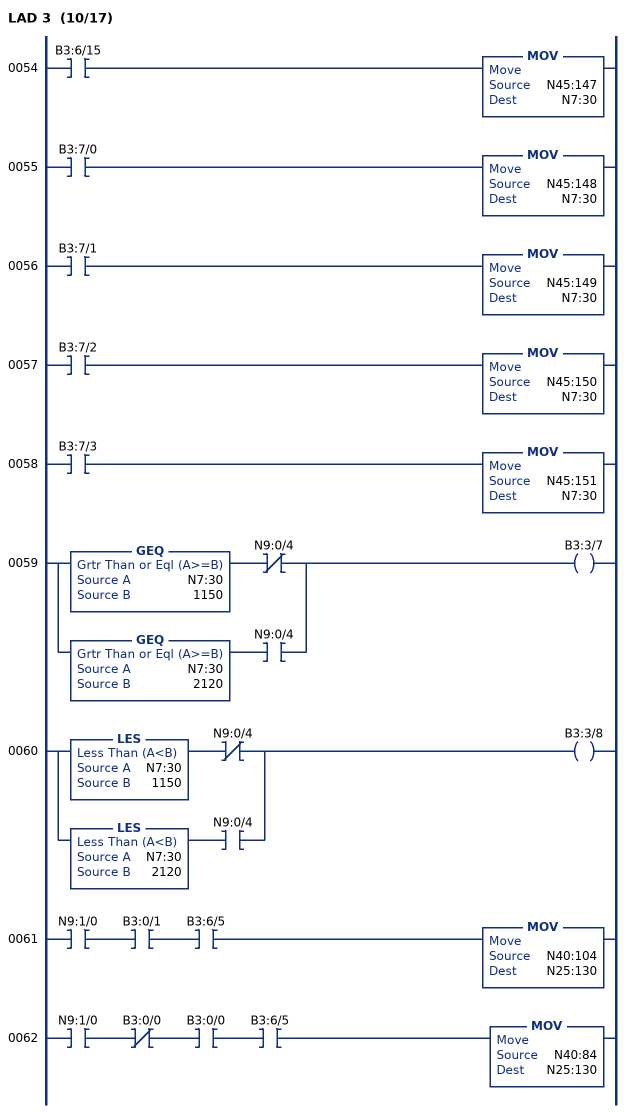
% Rung: 54 %
SOR XIC B3:6/15 MOV N45:147 N7:30 EOR
% Rung: 55 %
SOR XIC B3:7/0 MOV N45:148 N7:30 EOR
% Rung: 56 %
SOR XIC B3:7/1 MOV N45:149 N7:30 EOR
% Rung: 57 %
SOR XIC B3:7/2 MOV N45:150 N7:30 EOR
% Rung: 58 %
SOR XIC B3:7/3 MOV N45:151 N7:30 EOR
% Rung: 59 %
SOR BST GEQ N7:30 1150 XIO N9:0/4 NXB GEQ N7:30 2120 XIC N9:0/4 BND OTE B3:3/7 EOR
% Rung: 60 %
SOR BST LES N7:30 1150 XIO N9:0/4 NXB LES N7:30 2120 XIC N9:0/4 BND OTE B3:3/8 EOR
% Rung: 61 %
SOR XIC N9:1/0 XIC B3:0/1 XIC B3:6/5 MOV N40:104 N25:130 EOR
% Rung: 62 %
SOR XIC N9:1/0 XIO B3:0/0 XIC B3:0/0 XIC B3:6/5 MOV N40:84 N25:130 EOR

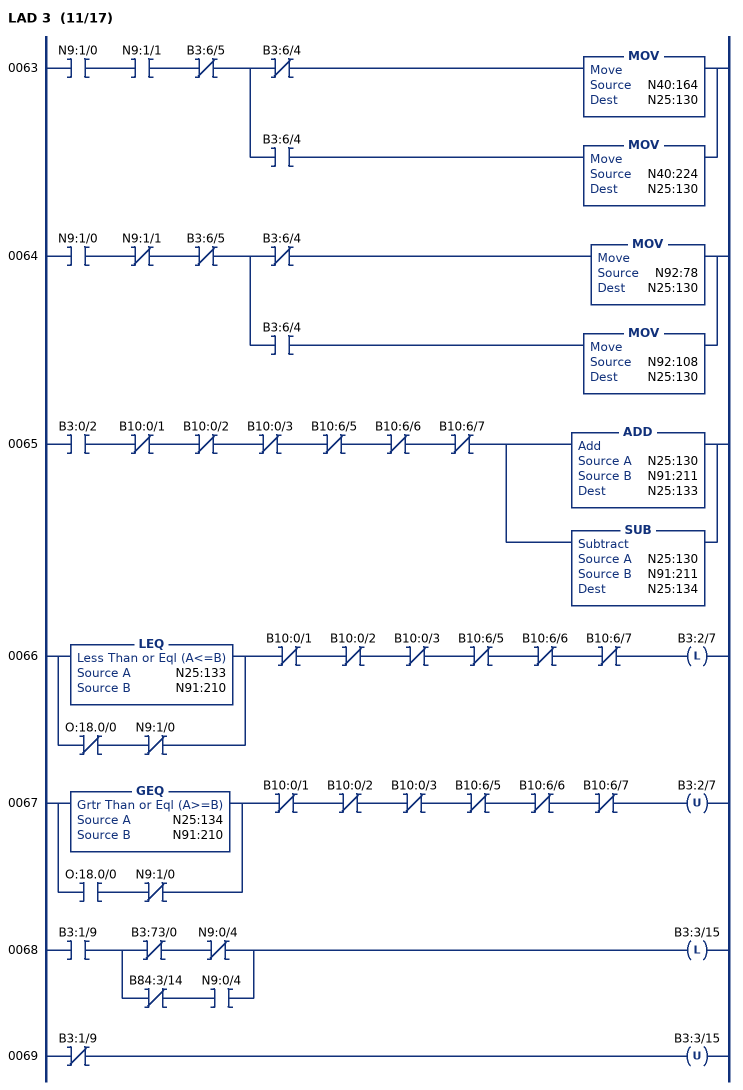
% Rung: 63 %
SOR XIC N9:1/0 XIC N9:1/1 XIO B3:6/5 BST XIO B3:6/4 MOV N40:164 N25:130 NXB XIC B3:6/4 MOV N40:224 N25:130 BND EOR
% Rung: 64 %
SOR XIC N9:1/0 XIO N9:1/1 XIO B3:6/5 BST XIO B3:6/4 MOV N92:78 N25:130 NXB XIC B3:6/4 MOV N92:108 N25:130 BND EOR
% Rung: 65 %
SOR XIC B3:0/2 XIO B10:0/1 XIO B10:0/2 XIO B10:0/3 XIO B10:6/5 XIO B10:6/6 XIO B10:6/7 BST ADD N25:130 N91:211 N25:133 NXB SUB N25:130 N91:211 N25:134 BND EOR
% Rung: 66 %
SOR BST LEQ N25:133 N91:210 NXB XIO O:18.0/0 XIO N9:1/0 BND XIO B10:0/1 XIO B10:0/2 XIO B10:0/3 XIO B10:6/5 XIO B10:6/6 XIO B10:6/7 OTL B3:2/7 EOR
% Rung: 67 %
SOR BST GEQ N25:134 N91:210 NXB XIC O:18.0/0 XIO N9:1/0 BND XIO B10:0/1 XIO B10:0/2 XIO B10:0/3 XIO B10:6/5 XIO B10:6/6 XIO B10:6/7 OTU B3:2/7 EOR
% Rung: 68 %
SOR XIC B3:1/9 BST XIO B3:73/0 XIO N9:0/4 NXB XIO B84:3/14 XIC N9:0/4 BND OTL B3:3/15 EOR
% Rung: 69 %
SOR XIO B3:1/9 OTU B3:3/15 EOR

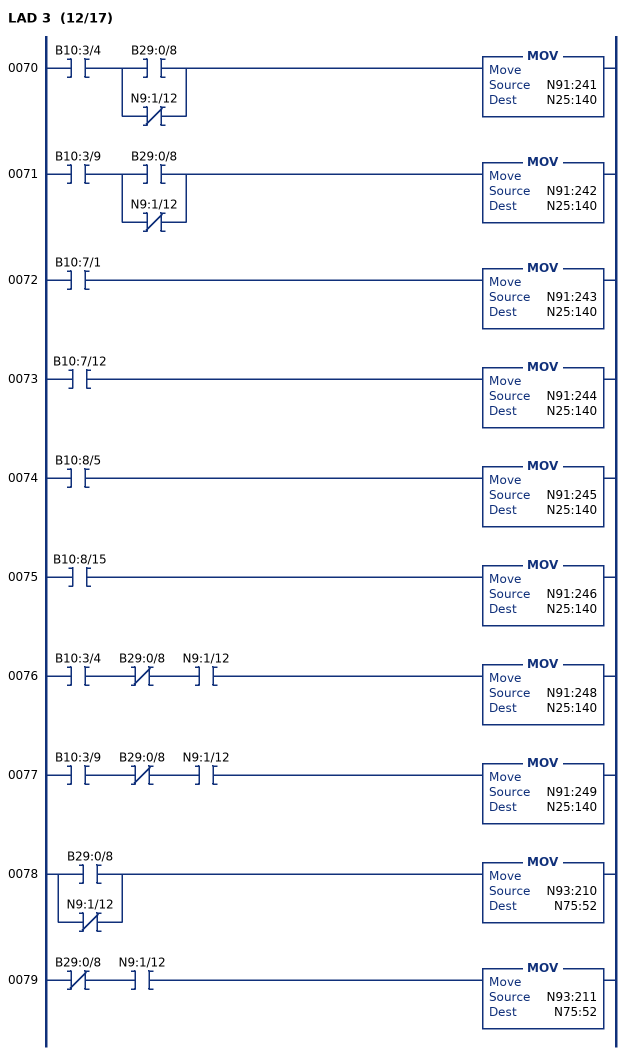
% Rung: 70 %
SOR XIC B10:3/4 BST XIC B29:0/8 NXB XIO N9:1/12 BND MOV N91:241 N25:140 EOR
% Rung: 71 %
SOR XIC B10:3/9 BST XIC B29:0/8 NXB XIO N9:1/12 BND MOV N91:242 N25:140 EOR
% Rung: 72 %
SOR XIC B10:7/1 MOV N91:243 N25:140 EOR
% Rung: 73 %
SOR XIC B10:7/12 MOV N91:244 N25:140 EOR
% Rung: 74 %
SOR XIC B10:8/5 MOV N91:245 N25:140 EOR
% Rung: 75 %
SOR XIC B10:8/15 MOV N91:246 N25:140 EOR
% Rung: 76 %
SOR XIC B10:3/4 XIO B29:0/8 XIC N9:1/12 MOV N91:248 N25:140 EOR
% Rung: 77 %
SOR XIC B10:3/9 XIO B29:0/8 XIC N9:1/12 MOV N91:249 N25:140 EOR
% Rung: 78 %
SOR BST XIC B29:0/8 NXB XIO N9:1/12 BND MOV N93:210 N75:52 EOR
% Rung: 79 %
SOR XIO B29:0/8 XIC N9:1/12 MOV N93:211 N75:52 EOR

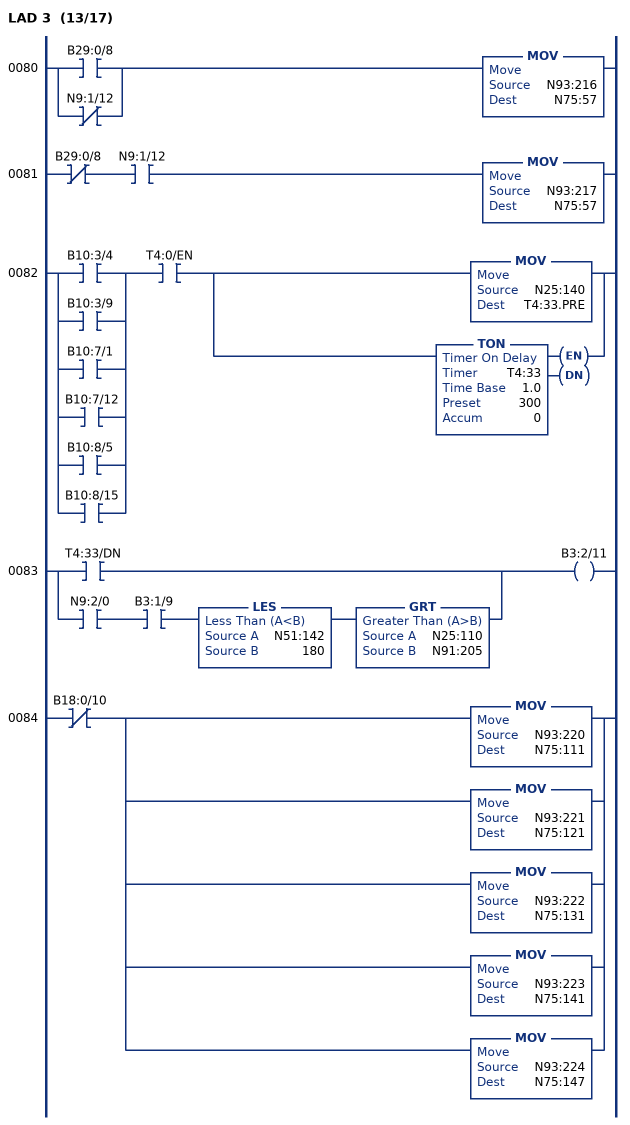
% Rung: 80 %
SOR BST XIC B29:0/8 NXB XIO N9:1/12 BND MOV N93:216 N75:57 EOR
% Rung: 81 %
SOR XIO B29:0/8 XIC N9:1/12 MOV N93:217 N75:57 EOR
% Rung: 82 %
SOR BST XIC B10:3/4 NXB XIC B10:3/9 NXB XIC B10:7/1 NXB XIC B10:7/12 NXB XIC B10:8/5 NXB XIC B10:8/15 BND XIC T4:0/EN BST MOV N25:140 T4:33.PRE NXB TON T4:33 1.0 300 0 BND EOR
% Rung: 83 %
SOR BST XIC T4:33/DN NXB XIC N9:2/0 XIC B3:1/9 LES N51:142 180 GRT N25:110 N91:205 BND OTE B3:2/11 EOR
% Rung: 84 %
SOR XIO B18:0/10 BST MOV N93:220 N75:111 NXB MOV N93:221 N75:121 NXB MOV N93:222 N75:131 NXB MOV N93:223 N75:141 NXB MOV N93:224 N75:147 BND EOR

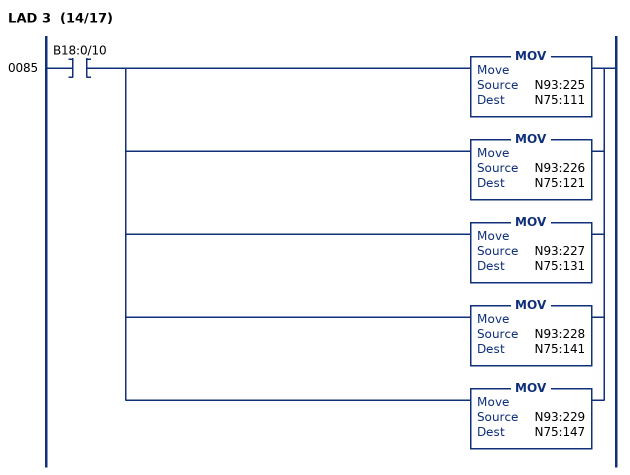
% Rung: 85 %
SOR XIC B18:0/10 BST MOV N93:225 N75:111 NXB MOV N93:226 N75:121 NXB MOV N93:227 N75:131 NXB MOV N93:228 N75:141 NXB MOV N93:229 N75:147 BND EOR

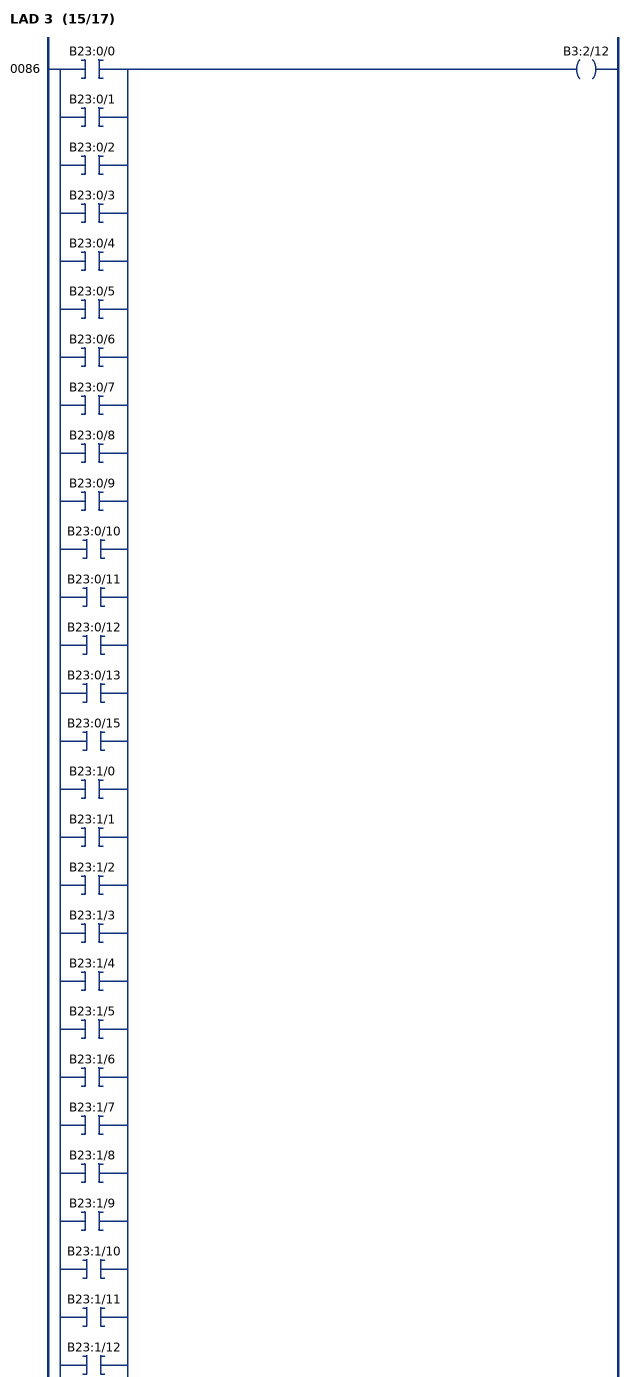

